FUNCTION_BLOCK Test_TStreamAdd_Read_INT_CheckAlignment EXTENDS T_UnitTestBase
VAR
    Stream  : T_Stream(StreamLength := 2);
    ArgType : E_ArgTypeId := E_ArgTypeId.Type_INT;
END_VAR

{attribute 'analysis' := '-33'} // inhibit unused variable warning
METHOD RunTest
Stream.Init(2);

Stream.Add_BYTE(123);// add a byte to test alignment checks...
Stream.Add_INT(1234);

Stream.SetReadPosition(0);

Stream.Read_BYTE();

// check next value...	
AssertEquals_INT(Expected     := 1234,
                           Actual       := Stream.Read_INT(),
                           Message := 'Stream.Read_INT()');

// check we are at the end of the stream..							
AssertEquals_UDINT(Expected     := Stream.StreamLength,
                             Actual       := Stream.ReadPosition,
                             Message := 'Stream.ReadPosition');

TestCompleted := TRUE;
END_METHOD

END_FUNCTION_BLOCK

(* stored: Version 1.1.0.1, ProductVersion 3.1.4024.12
   POU Test_TStreamAdd_Read_INT_CheckAlignment: Id {e45de268-e5ec-4062-a160-f2f860e4df85}, SpecialFunc None
   Method RunTest: Id {486c8cfa-7623-4db8-85f0-979dc7b5f859} *)
